// TIA Portal V19 export
VAR_GLOBAL   // PLC tag table "U2Em2Output"
   "null(8)" AT %Q42.4 : Bool;   // 备用
   "null(10)" AT %Q42.6 : Bool;   // 备用
   "null(6)" AT %Q42.2 : Bool;   // 备用
   "null(13)" AT %Q43.3 : Bool;   // 备用
   cellLiftingCylinderWorkPositionU2Em2 AT %Q43.0 : Bool;   // U2Em2_Battery lifting cylinder working position / Em90_电池升降气缸工作位
   trayLiftingCylinderWorkPositionU2Em2 AT %Q42.0 : Bool;   // U2Em2_ pallet lifting cylinder working position / Em90_托盘顶升气缸工作位
   positioningPinCylinderWorkingPositionU2Em2_1 AT %Q43.4 : Bool;   // U2Em2_Positioning Pin Cylinder 1 Working Position / Em90_定位销气缸1工作位
   positioningPinCylinderHomePositionU2Em2_1 AT %Q43.5 : Bool;   // U2Em2_Positioning Pin Cylinder 1 Home Position / Em90_定位销气缸1原位
   trayLiftingCylinderHomePositionU2Em2 AT %Q42.1 : Bool;   // U2Em2_Tray Jacking Cylinder Home Position / Em90_托盘顶升气缸原位
   cellLiftingCylinderHomePositionU2Em2 AT %Q43.1 : Bool;   // U2Em2_Battery Lift Cylinder Home Position / Em90_电池升降气缸原位
   "null(12)" AT %Q43.2 : Bool;   // spare / 备用
   "null(11)" AT %Q42.7 : Bool;   // spare / 备用
   "null(9)" AT %Q42.5 : Bool;   // spare / 备用
   "null(7)" AT %Q42.3 : Bool;   // spare / 备用
END_VAR
